TYPE ST_PressureInputScaling :
STRUCT
	fMaxInputValue 			: LREAL;	// tunable max input value 
	fMinInputValue			: LREAL;	// tunable min input value  
	fMaxOutputValue  		: LREAL;	// max sensor output value
	fMinOutputValue  		: LREAL;	// min sensor output value	
END_STRUCT
END_TYPE

(* stored: Version 1.1.0.1
   DUT ST_PressureInputScaling: Id {1701137f-c4b2-4ef2-b379-08d42d80a31e} *)
